{attribute 'qualified_only'}
{attribute 'strict'}
TYPE e_controllerStatus :
(
	None 	:= 	0,
	Init	:=	1,
	Ready	:=	2,
	Active	:=	3,
	Error	:=	4
);
END_TYPE

(* stored: Version 1.1.0.1, ProductVersion 3.1.4024.12
   DUT e_controllerStatus: Id {b2792a1a-243b-4f73-b333-eea7ed0aebf9} *)
